// TIA Portal V19 export
TYPE "LubrValve_Alr"
// stored: Access Published
   STRUCT
      CycleFeedback : Bool;   // Cycle feedback not engaged during lubrication
      ConnectorNotPlugged : Bool;
      ConfigError : Bool;   // Check config of valve
   END_STRUCT;
END_TYPE
